{attribute 'qualified_only'}
VAR_GLOBAL
	fJoystickLeftNormalizedY 		: LREAL;
	fJoystickLeftNormalizedX 		: LREAL;	
	fJoystickRightNormalizedY 		: LREAL;
	fJoystickRightNormalizedX 		: LREAL;
	
	nJoystickLeftDirectionX 		: DINT;
	nJoystickLeftDirectionY 		: DINT;
	nJoystickRightDirectionX 		: DINT;
	nJoystickRightDirectionY 		: DINT;
	
	bJoystick1InUse : BOOL ;
	bJoystick2InUse : BOOL;
	bJoystick3InUse : BOOL;
	bJoystick4InUse : BOOL;
		
END_VAR

(* stored: Version 1.1.0.1, ProductVersion 3.1.4024.12
   GVL G_Joystick: Id {c722b76a-a2a7-461a-a024-0641a38117f7} *)
